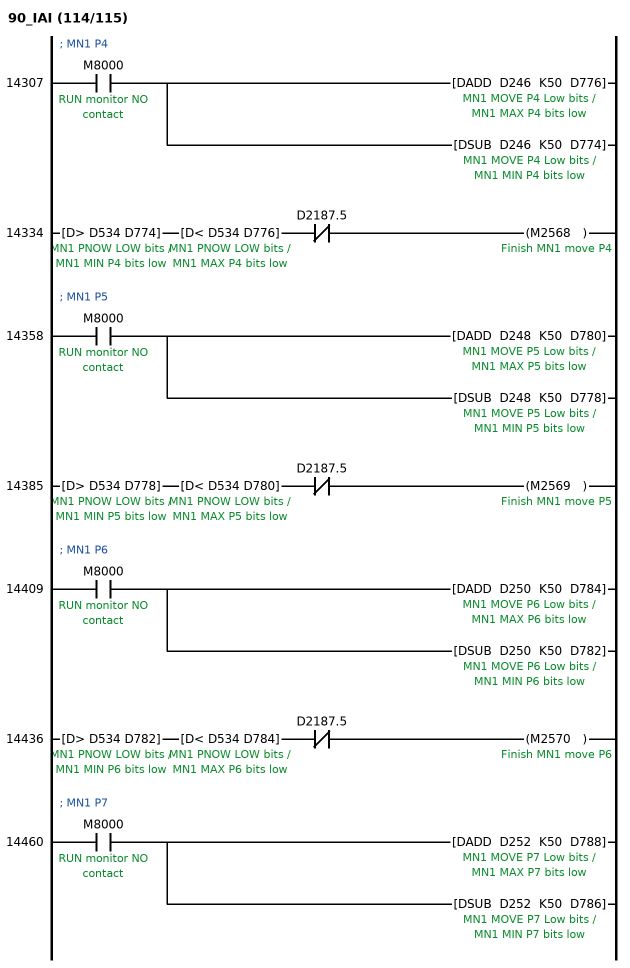
[picture p216: ladder of 90_IAI, rungs at steps 14307 to 14460]
; MN1 P4
14307 LD      M8000  ; RUN monitor NO contact
      DADD    D246 K50 D776  ; MN1 MAX P4 bits low
      DSUB    D246 K50 D774  ; MN1 MIN P4 bits low
14334 LDD>    D534 D774  ; MN1 PNOW LOW bits / MN1 MIN P4 bits low
      ANDD<   D534 D776  ; MN1 PNOW LOW bits / MN1 MAX P4 bits low
      ANI     D2187.5
      OUT     M2568  ; Finish MN1 move P4
; MN1 P5
14358 LD      M8000  ; RUN monitor NO contact
      DADD    D248 K50 D780  ; MN1 MAX P5 bits low
      DSUB    D248 K50 D778  ; MN1 MIN P5 bits low
14385 LDD>    D534 D778  ; MN1 PNOW LOW bits / MN1 MIN P5 bits low
      ANDD<   D534 D780  ; MN1 PNOW LOW bits / MN1 MAX P5 bits low
      ANI     D2187.5
      OUT     M2569  ; Finish MN1 move P5
; MN1 P6
14409 LD      M8000  ; RUN monitor NO contact
      DADD    D250 K50 D784  ; MN1 MAX P6 bits low
      DSUB    D250 K50 D782  ; MN1 MIN P6 bits low
14436 LDD>    D534 D782  ; MN1 PNOW LOW bits / MN1 MIN P6 bits low
      ANDD<   D534 D784  ; MN1 PNOW LOW bits / MN1 MAX P6 bits low
      ANI     D2187.5
      OUT     M2570  ; Finish MN1 move P6
; MN1 P7
14460 LD      M8000  ; RUN monitor NO contact
      DADD    D252 K50 D788  ; MN1 MAX P7 bits low
      DSUB    D252 K50 D786  ; MN1 MIN P7 bits low
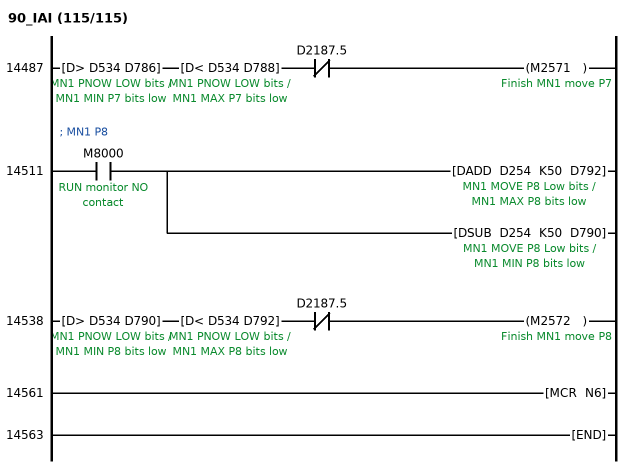
14487 LDD>    D534 D786  ; MN1 PNOW LOW bits / MN1 MIN P7 bits low
      ANDD<   D534 D788  ; MN1 PNOW LOW bits / MN1 MAX P7 bits low
      ANI     D2187.5
      OUT     M2571  ; Finish MN1 move P7
; MN1 P8
14511 LD      M8000  ; RUN monitor NO contact
      DADD    D254 K50 D792  ; MN1 MAX P8 bits low
      DSUB    D254 K50 D790  ; MN1 MIN P8 bits low
14538 LDD>    D534 D790  ; MN1 PNOW LOW bits / MN1 MIN P8 bits low
      ANDD<   D534 D792  ; MN1 PNOW LOW bits / MN1 MAX P8 bits low
      ANI     D2187.5
      OUT     M2572  ; Finish MN1 move P8
14561 MCR     N6
14563 END
END_PROGRAM

PROGRAM 91_Pr_Te
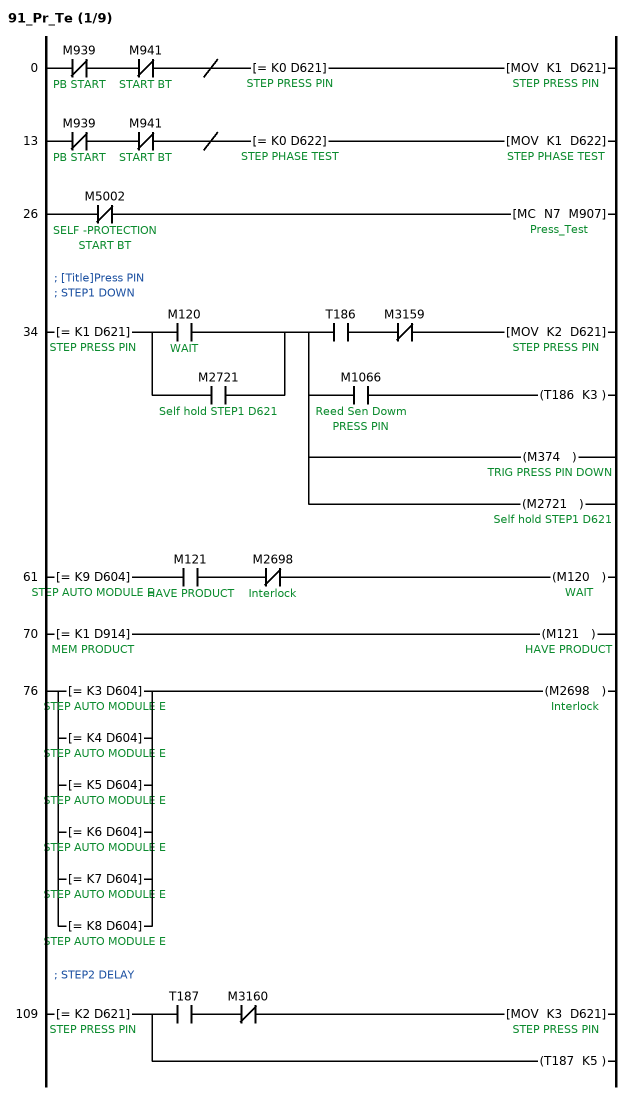
0     LDI     M939  ; PB START
      ANI     M941  ; START BT
      INV
      AND=    K0 D621  ; STEP PRESS PIN
      MOV     K1 D621
13    LDI     M939  ; PB START
      ANI     M941  ; START BT
      INV
      AND=    K0 D622  ; STEP PHASE TEST
      MOV     K1 D622
26    LDI     M5002  ; SELF -PROTECTION START BT
      MC      N7 M907  ; Press_Test
; [Title]Press PIN
; STEP1 DOWN
34    LD=     K1 D621  ; STEP PRESS PIN
      LD      M120  ; WAIT
      OR      M2721  ; Self hold STEP1 D621
      ANB
      MPS
      AND     T186
      ANI     M3159
      MOV     K2 D621
      MRD
      AND     M1066  ; Reed Sen Dowm PRESS PIN
      OUT     T186 K3
      MPP
      OUT     M374  ; TRIG PRESS PIN DOWN
      OUT     M2721  ; Self hold STEP1 D621
61    LD=     K9 D604  ; STEP AUTO MODULE E
      AND     M121  ; HAVE PRODUCT
      ANI     M2698  ; Interlock
      OUT     M120  ; WAIT
70    LD=     K1 D914  ; MEM PRODUCT
      OUT     M121  ; HAVE PRODUCT
76    LD=     K3 D604  ; STEP AUTO MODULE E
      OR=     K4 D604  ; STEP AUTO MODULE E
      OR=     K5 D604  ; STEP AUTO MODULE E
      OR=     K6 D604  ; STEP AUTO MODULE E
      OR=     K7 D604  ; STEP AUTO MODULE E
      OR=     K8 D604  ; STEP AUTO MODULE E
      OUT     M2698  ; Interlock
; STEP2 DELAY
109   LD=     K2 D621  ; STEP PRESS PIN
      MPS
      AND     T187
      ANI     M3160
      MOV     K3 D621
      MPP
      OUT     T187 K5
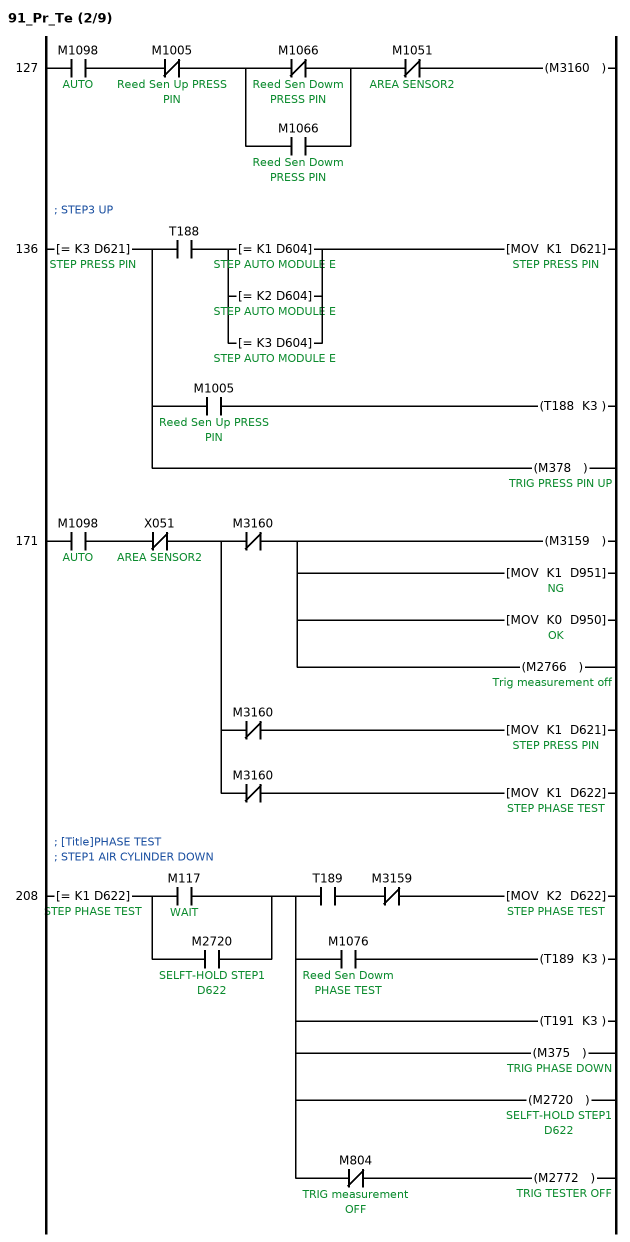
127   LD      M1098  ; AUTO
      ANI     M1005  ; Reed Sen Up PRESS PIN
      LDI     M1066  ; Reed Sen Dowm PRESS PIN
      OR      M1066  ; Reed Sen Dowm PRESS PIN
      ANB
      ANI     M1051  ; AREA SENSOR2
      OUT     M3160
; STEP3 UP
136   LD=     K3 D621  ; STEP PRESS PIN
      MPS
      AND     T188
      LD=     K1 D604  ; STEP AUTO MODULE E
      OR=     K2 D604  ; STEP AUTO MODULE E
      OR=     K3 D604  ; STEP AUTO MODULE E
      ANB
      MOV     K1 D621
      MRD
      AND     M1005  ; Reed Sen Up PRESS PIN
      OUT     T188 K3
      MPP
      OUT     M378  ; TRIG PRESS PIN UP
171   LD      M1098  ; AUTO
      ANI     X051  ; AREA SENSOR2
      MPS
      ANI     M3160
      OUT     M3159
      MOV     K1 D951  ; NG
      MOV     K0 D950  ; OK
      OUT     M2766  ; Trig measurement off
      MRD
      ANI     M3160
      MOV     K1 D621
      MPP
      ANI     M3160
      MOV     K1 D622
; [Title]PHASE TEST
; STEP1 AIR CYLINDER DOWN
208   LD=     K1 D622  ; STEP PHASE TEST
      LD      M117  ; WAIT
      OR      M2720  ; SELFT-HOLD STEP1 D622
      ANB
      MPS
      AND     T189
      ANI     M3159
      MOV     K2 D622
      MRD
      AND     M1076  ; Reed Sen Dowm PHASE TEST
      OUT     T189 K3
      MPP
      OUT     T191 K3
      OUT     M375  ; TRIG PHASE DOWN
      OUT     M2720  ; SELFT-HOLD STEP1 D622
      ANI     M804  ; TRIG measurement OFF
      OUT     M2772  ; TRIG TESTER OFF
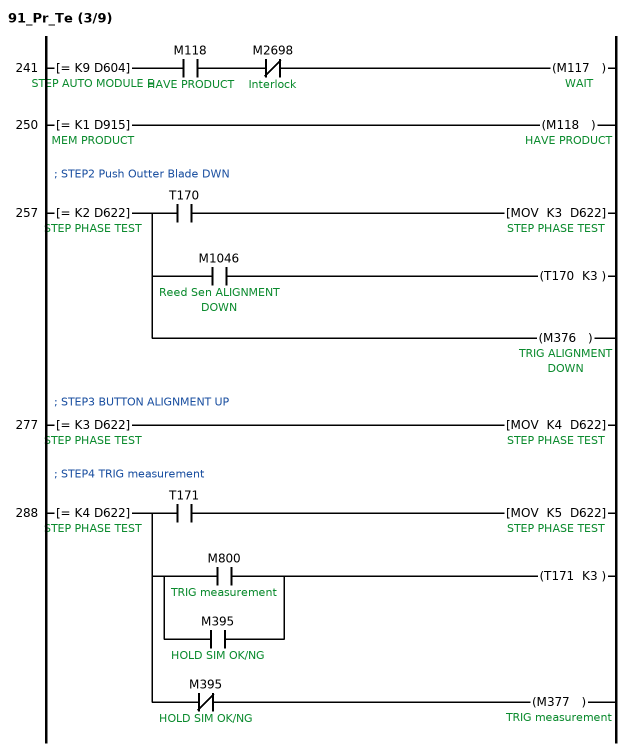
241   LD=     K9 D604  ; STEP AUTO MODULE E
      AND     M118  ; HAVE PRODUCT
      ANI     M2698  ; Interlock
      OUT     M117  ; WAIT
250   LD=     K1 D915  ; MEM PRODUCT
      OUT     M118  ; HAVE PRODUCT
; STEP2 Push Outter Blade DWN
257   LD=     K2 D622  ; STEP PHASE TEST
      MPS
      AND     T170
      MOV     K3 D622
      MRD
      AND     M1046  ; Reed Sen ALIGNMENT DOWN
      OUT     T170 K3
      MPP
      OUT     M376  ; TRIG ALIGNMENT DOWN
; STEP3 BUTTON ALIGNMENT UP
277   LD=     K3 D622  ; STEP PHASE TEST
      MOV     K4 D622
; STEP4 TRIG measurement
288   LD=     K4 D622  ; STEP PHASE TEST
      MPS
      AND     T171
      MOV     K5 D622
      MRD
      LD      M800  ; TRIG measurement
      OR      M395  ; HOLD SIM OK/NG
      ANB
      OUT     T171 K3
      MPP
      ANI     M395  ; HOLD SIM OK/NG
      OUT     M377  ; TRIG measurement
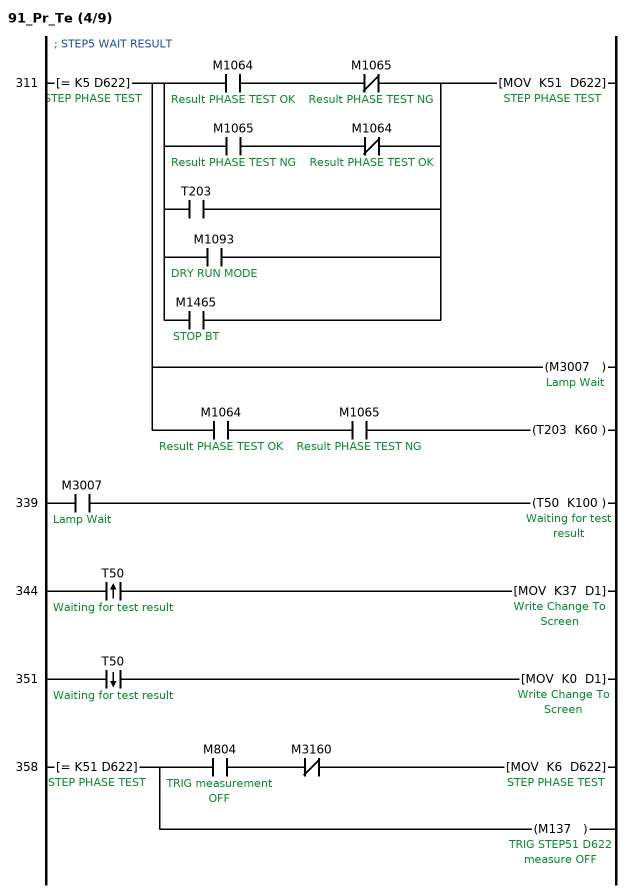
; STEP5 WAIT RESULT
311   LD=     K5 D622  ; STEP PHASE TEST
      MPS
      LD      M1064  ; Result PHASE TEST OK
      ANI     M1065  ; Result PHASE TEST NG
      LD      M1065  ; Result PHASE TEST NG
      ANI     M1064  ; Result PHASE TEST OK
      ORB
      OR      T203
      OR      M1093  ; DRY RUN MODE
      OR      M1465  ; STOP BT
      ANB
      MOV     K51 D622
      MPP
      OUT     M3007  ; Lamp Wait
      AND     M1064  ; Result PHASE TEST OK
      AND     M1065  ; Result PHASE TEST NG
      OUT     T203 K60
339   LD      M3007  ; Lamp Wait
      OUT     T50 K100  ; Waiting for test result
344   LDP     T50  ; Waiting for test result
      MOV     K37 D1  ; Write Change To Screen
351   LDF     T50  ; Waiting for test result
      MOV     K0 D1
358   LD=     K51 D622  ; STEP PHASE TEST
      MPS
      AND     M804  ; TRIG measurement OFF
      ANI     M3160
      MOV     K6 D622
      MPP
      OUT     M137  ; TRIG STEP51 D622 measure OFF
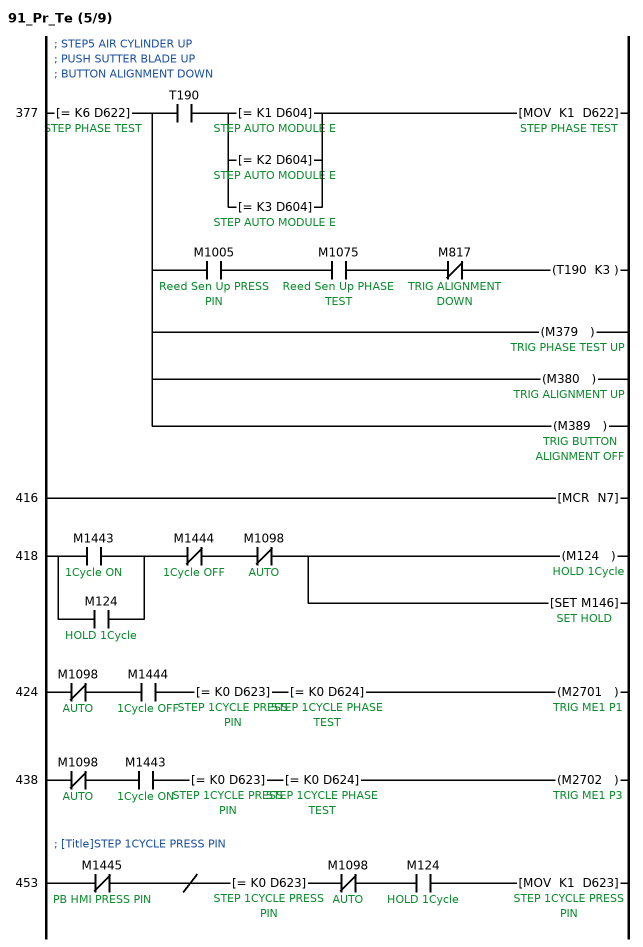
; STEP5 AIR CYLINDER UP
; PUSH SUTTER BLADE UP
; BUTTON ALIGNMENT DOWN
377   LD=     K6 D622  ; STEP PHASE TEST
      MPS
      AND     T190
      LD=     K1 D604  ; STEP AUTO MODULE E
      OR=     K2 D604  ; STEP AUTO MODULE E
      OR=     K3 D604  ; STEP AUTO MODULE E
      ANB
      MOV     K1 D622
      MRD
      AND     M1005  ; Reed Sen Up PRESS PIN
      AND     M1075  ; Reed Sen Up PHASE TEST
      ANI     M817  ; TRIG ALIGNMENT  DOWN
      OUT     T190 K3
      MPP
      OUT     M379  ; TRIG PHASE TEST UP
      OUT     M380  ; TRIG ALIGNMENT UP
      OUT     M389  ; TRIG BUTTON ALIGNMENT OFF
416   MCR     N7
418   LD      M1443  ; 1Cycle ON
      OR      M124  ; HOLD 1Cycle
      ANI     M1444  ; 1Cycle OFF
      ANI     M1098  ; AUTO
      OUT     M124  ; HOLD 1Cycle
      SET     M146  ; SET HOLD
424   LDI     M1098  ; AUTO
      AND     M1444  ; 1Cycle OFF
      AND=    K0 D623  ; STEP 1CYCLE PRESS PIN
      AND=    K0 D624  ; STEP 1CYCLE PHASE TEST
      OUT     M2701  ; TRIG ME1 P1
438   LDI     M1098  ; AUTO
      AND     M1443  ; 1Cycle ON
      AND=    K0 D623  ; STEP 1CYCLE PRESS PIN
      AND=    K0 D624  ; STEP 1CYCLE PHASE TEST
      OUT     M2702  ; TRIG ME1 P3
; [Title]STEP 1CYCLE PRESS PIN
453   LDI     M1445  ; PB HMI PRESS PIN
      INV
      AND=    K0 D623  ; STEP 1CYCLE PRESS PIN
      ANI     M1098  ; AUTO
      AND     M124  ; HOLD 1Cycle
      MOV     K1 D623
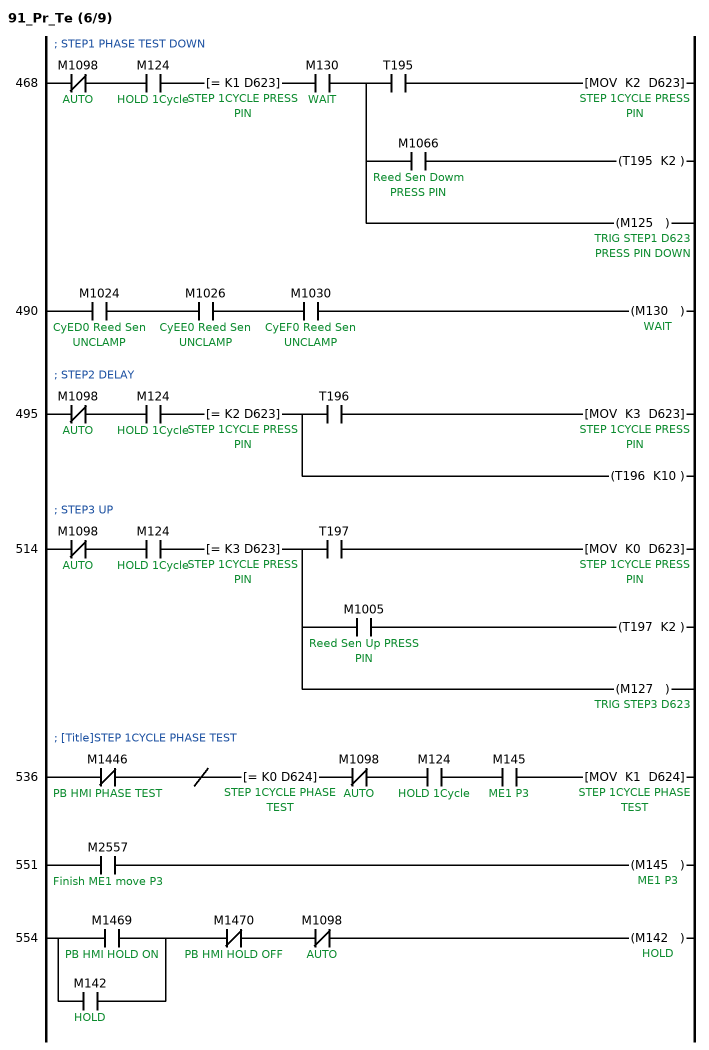
; STEP1 PHASE TEST DOWN
468   LDI     M1098  ; AUTO
      AND     M124  ; HOLD 1Cycle
      AND=    K1 D623  ; STEP 1CYCLE PRESS PIN
      AND     M130  ; WAIT
      MPS
      AND     T195
      MOV     K2 D623
      MRD
      AND     M1066  ; Reed Sen Dowm PRESS PIN
      OUT     T195 K2
      MPP
      OUT     M125  ; TRIG STEP1 D623 PRESS PIN DOWN
490   LD      M1024  ; CyED0 Reed Sen UNCLAMP
      AND     M1026  ; CyEE0 Reed Sen UNCLAMP
      AND     M1030  ; CyEF0 Reed Sen UNCLAMP
      OUT     M130  ; WAIT
; STEP2 DELAY
495   LDI     M1098  ; AUTO
      AND     M124  ; HOLD 1Cycle
      AND=    K2 D623  ; STEP 1CYCLE PRESS PIN
      MPS
      AND     T196
      MOV     K3 D623
      MPP
      OUT     T196 K10
; STEP3 UP
514   LDI     M1098  ; AUTO
      AND     M124  ; HOLD 1Cycle
      AND=    K3 D623  ; STEP 1CYCLE PRESS PIN
      MPS
      AND     T197
      MOV     K0 D623
      MRD
      AND     M1005  ; Reed Sen Up PRESS PIN
      OUT     T197 K2
      MPP
      OUT     M127  ; TRIG STEP3 D623
; [Title]STEP 1CYCLE PHASE TEST
536   LDI     M1446  ; PB HMI PHASE TEST
      INV
      AND=    K0 D624  ; STEP 1CYCLE PHASE TEST
      ANI     M1098  ; AUTO
      AND     M124  ; HOLD 1Cycle
      AND     M145  ; ME1 P3
      MOV     K1 D624
551   LD      M2557  ; Finish ME1 move P3
      OUT     M145  ; ME1 P3
554   LD      M1469  ; PB HMI HOLD ON
      OR      M142  ; HOLD
      ANI     M1470  ; PB HMI HOLD OFF
      ANI     M1098  ; AUTO
      OUT     M142  ; HOLD
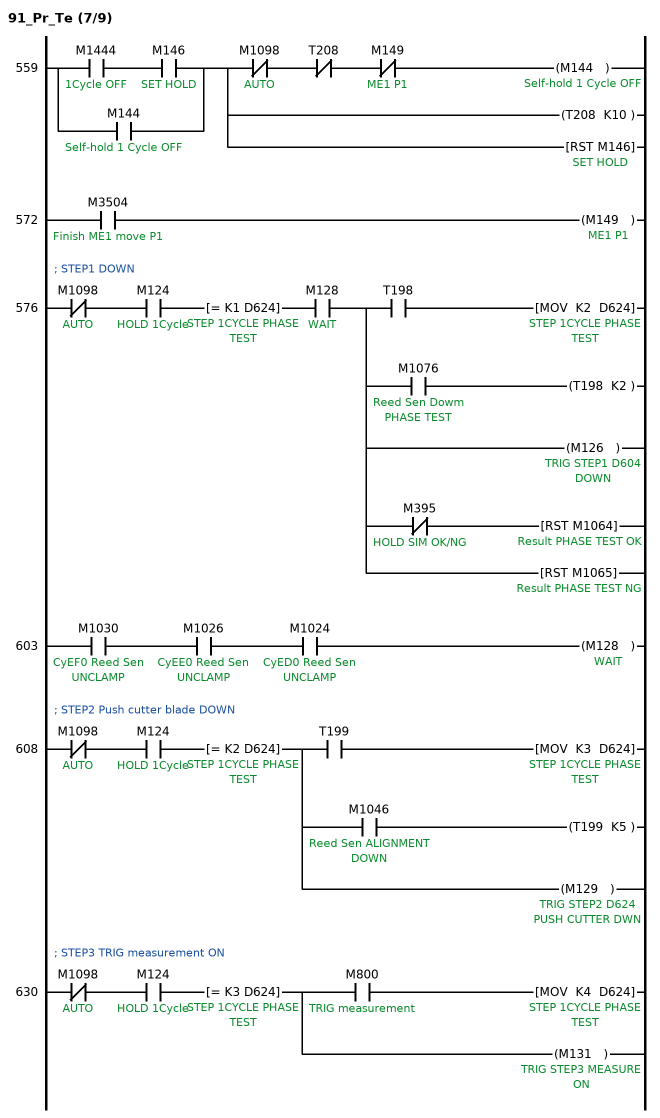
559   LD      M1444  ; 1Cycle OFF
      AND     M146  ; SET HOLD
      OR      M144  ; Self-hold 1 Cycle OFF
      MPS
      ANI     M1098  ; AUTO
      ANI     T208
      ANI     M149  ; ME1 P1
      OUT     M144  ; Self-hold 1 Cycle OFF
      MPP
      OUT     T208 K10
      RST     M146  ; SET HOLD
572   LD      M3504  ; Finish ME1 move P1
      OUT     M149  ; ME1 P1
; STEP1 DOWN
576   LDI     M1098  ; AUTO
      AND     M124  ; HOLD 1Cycle
      AND=    K1 D624  ; STEP 1CYCLE PHASE TEST
      AND     M128  ; WAIT
      MPS
      AND     T198
      MOV     K2 D624
      MRD
      AND     M1076  ; Reed Sen Dowm PHASE TEST
      OUT     T198 K2
      MPP
      OUT     M126  ; TRIG STEP1 D604 DOWN
      MPS
      ANI     M395  ; HOLD SIM OK/NG
      RST     M1064  ; Result PHASE TEST OK
      MPP
      RST     M1065  ; Result PHASE TEST NG
603   LD      M1030  ; CyEF0 Reed Sen UNCLAMP
      AND     M1026  ; CyEE0 Reed Sen UNCLAMP
      AND     M1024  ; CyED0 Reed Sen UNCLAMP
      OUT     M128  ; WAIT
; STEP2 Push cutter blade DOWN
608   LDI     M1098  ; AUTO
      AND     M124  ; HOLD 1Cycle
      AND=    K2 D624  ; STEP 1CYCLE PHASE TEST
      MPS
      AND     T199
      MOV     K3 D624
      MRD
      AND     M1046  ; Reed Sen ALIGNMENT DOWN
      OUT     T199 K5
      MPP
      OUT     M129  ; TRIG STEP2 D624 PUSH CUTTER DWN
; STEP3 TRIG measurement ON
630   LDI     M1098  ; AUTO
      AND     M124  ; HOLD 1Cycle
      AND=    K3 D624  ; STEP 1CYCLE PHASE TEST
      MPS
      AND     M800  ; TRIG measurement
      MOV     K4 D624
      MPP
      OUT     M131  ; TRIG STEP3 MEASURE ON
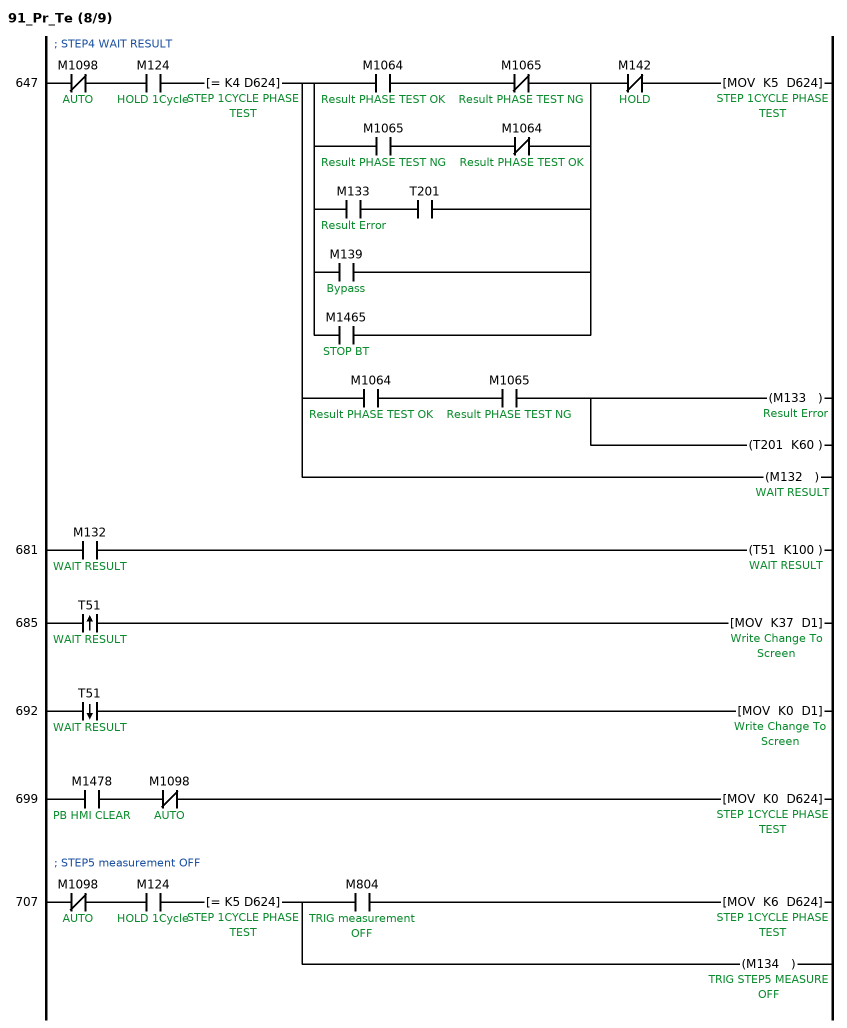
; STEP4 WAIT RESULT
647   LDI     M1098  ; AUTO
      AND     M124  ; HOLD 1Cycle
      AND=    K4 D624  ; STEP 1CYCLE PHASE TEST
      MPS
      LD      M1064  ; Result PHASE TEST OK
      ANI     M1065  ; Result PHASE TEST NG
      LD      M1065  ; Result PHASE TEST NG
      ANI     M1064  ; Result PHASE TEST OK
      ORB
      LD      M133  ; Result Error
      AND     T201
      ORB
      OR      M139  ; Bypass
      OR      M1465  ; STOP BT
      ANB
      ANI     M142  ; HOLD
      MOV     K5 D624
      MRD
      AND     M1064  ; Result PHASE TEST OK
      AND     M1065  ; Result PHASE TEST NG
      OUT     M133  ; Result Error
      OUT     T201 K60
      MPP
      OUT     M132  ; WAIT RESULT
681   LD      M132  ; WAIT RESULT
      OUT     T51 K100  ; WAIT RESULT
685   LDP     T51  ; WAIT RESULT
      MOV     K37 D1
692   LDF     T51  ; WAIT RESULT
      MOV     K0 D1
699   LD      M1478  ; PB HMI CLEAR
      ANI     M1098  ; AUTO
      MOV     K0 D624
; STEP5 measurement OFF
707   LDI     M1098  ; AUTO
      AND     M124  ; HOLD 1Cycle
      AND=    K5 D624  ; STEP 1CYCLE PHASE TEST
      MPS
      AND     M804  ; TRIG measurement OFF
      MOV     K6 D624
      MPP
      OUT     M134  ; TRIG STEP5 MEASURE OFF
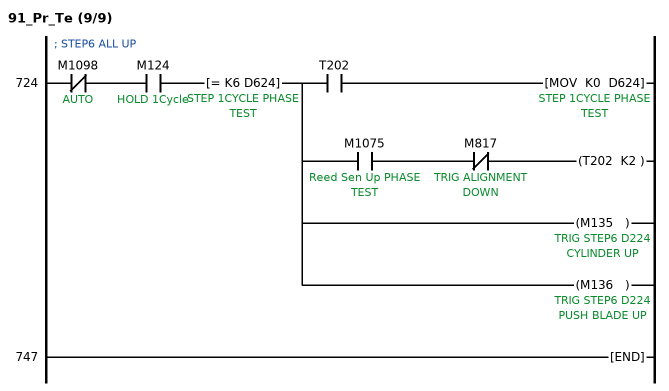
; STEP6 ALL UP
724   LDI     M1098  ; AUTO
      AND     M124  ; HOLD 1Cycle
      AND=    K6 D624  ; STEP 1CYCLE PHASE TEST
      MPS
      AND     T202
      MOV     K0 D624
      MRD
      AND     M1075  ; Reed Sen Up PHASE TEST
      ANI     M817  ; TRIG ALIGNMENT  DOWN
      OUT     T202 K2
      MPP
      OUT     M135  ; TRIG STEP6 D224 CYLINDER UP
      OUT     M136  ; TRIG STEP6 D224 PUSH BLADE UP
747   END
END_PROGRAM

// device comments not shown above
M147  ; ME1 P3
M480  ; 2
M676  ; MUTE LIGHT
M681  ; ALARM RESET
M1018  ; MC2_*ALM
M1048  ; ME1_HOME_OK
M1122  ; REED SW AIR GRIPPER
M1123  ; REED SW AIR GRIPPER
M1128  ; MB3_HOME_OK
M1129  ; MB3_SV
M1138  ; MB3_*ALM
M1148  ; ME1_HOME_OK [CON.2 OUT 14B]
M1149  ; ME1_SV
M1158  ; ME1_*ALM
M1159  ; ME1_HOME_OK SELF-PROTECTION
M1168  ; ALL IAI HOME_OK
M1206  ; TEST
M1217  ; HOME_OK ALL UNCLAMP
M1221  ; XIA = ON
M1222  ; XIB = ON
M1223  ; XIA = ON
M1300  ; HMI PB AIR GRIPPER CLAMP
M1301  ; HMI PB AIR GRIPPER UNCLAMP
M1310  ; PB HMI CyBG Down
M1311  ; PB HMI CyBG UP
M1314  ; PB HMI CyBF Clamp
M1315  ; PB HMI CyBF Unclamp
M1343  ; PB HMI SIDE1 [Y43]
M1406  ; MUTE
M1409  ; PB HMI START FLUX DIP
M1411  ; ALARM RESET
M1413  ; PB HMI RESET STEP HOME
M1418  ; PB HMI Start Flux 1 cycle
M1428  ; PB HMI START NG BLOCK
M1429  ; PB HMI RESTART CON.1
M1460  ; Bypass Result OK/NG ON
M1461  ; Bypass Result OK/NG OFF
M1462  ; HOME BT
M2000  ; PCON 8 AXIS SCAN1
M2001  ; Finsh Mov
M2002  ; Finish MOV
M2150  ; Finish Move
M2216  ; READ SLAVE1 MB1
M2217  ; READ SLAVE2 MB2
M2218  ; READ SLAVE3 MB3
M2219  ; READ SLAVE4 MC1
M2220  ; READ SLAVE5 MC2
M2221  ; READ SLAVE6 MD1
M2222  ; READ SLAVE7 ME1
M2223  ; READ SLAVE8 MN1
M3000  ; PCON 8 AXIS SCAN2
M3562  ; Finish STEP11 D601
M3563  ; Finish STEP12 D601
M4000  ; PCON 8 AXIS SCAN2
M5621  ; ST1 Slave1
M5622  ; ST2 Slave1
M5623  ; ST3 Slave1
M5624  ; ST4 Slave1
M5625  ; ST5 Slave1
M5626  ; ST6 Slave1
M5627  ; ST7 Slave1
M5628  ; JOG- Slave1
M5629  ; JOG+ Slave1
M5634  ; JISL Slave1
M5640  ; DRG1 Slave2
M5661  ; ST1 Slave2
M5662  ; ST2 Slave2
M5663  ; ST3 Slave2
M5664  ; ST4 Slave2
M5665  ; ST5 Slave2
M5666  ; ST6 Slave2
M5667  ; ST7 Slave2
M5668  ; JOG- Slave2
M5669  ; JOG+ Slave2
M5670  ; TEAC Slave2
M5671  ; MOD Slave2
M5674  ; JISL Slave2
M5701  ; ST1 Slave3
M5702  ; ST2 Slave3
M5703  ; ST3 Slave3
M5704  ; ST4 Slave3
M5705  ; ST5 Slave3
M5706  ; ST6 Slave3
M5707  ; ST7 Slave3
M5708  ; JOG- Slave3
M5709  ; JOG+ Slave3
M5714  ; JISL Slave3
M6001  ; Self-hold Bypass Solder Up/Down
D101  ; MB1 MOVE P1 Hight bits
D103  ; MB1 MOVE P2 Hight bits
D105  ; MB1 MOVE P3 Hight bits
D107  ; MB1 MOVE P4 Hight bits
D109  ; MB1 MOVE P5 Hight bits
D111  ; MB1 MOVE P6 Hight bits
D113  ; MB1 MOVE P7 Hight bits
D115  ; MB1 MOVE P8 Hight bits
D117  ; MB1 MOVE P9 Hight bits
D119  ; MB1 MOVE P10 Hight bits
D121  ; MB2 MOVE P1 Hight bits
D123  ; MB2 MOVE P2 Hight bits
D125  ; MB2 MOVE P3 Hight bits
D127  ; MB2 MOVE P4 Hight bits
D129  ; MB2 MOVE P5 Hight bits
D131  ; MB2 MOVE P6 Hight bits
D133  ; MB2 MOVE P7 Hight bits
D135  ; MB2 MOVE P8 Hight bits
D136  ; MB2 MOVE P9 Low bits
D137  ; MB2 MOVE P9 Hight bits
D138  ; MB2 MOVE P10 Low bits
D139  ; MB2 MOVE P10 Hight bits
D141  ; MB3 MOVE P1 Hight bits
D143  ; MB3 MOVE P2 Hight bits
D145  ; MB3 MOVE P3 Hight bits
D147  ; MB3 MOVE P4 Hight bits
D149  ; MB3 MOVE P5 Hight bits
D151  ; MB3 MOVE P6 Hight bits
D153  ; MB3 MOVE P7 Hight bits
D155  ; MB3 MOVE P8 Hight bits
D156  ; MB3 MOVE P9 Low bits
D157  ; MB3 MOVE P9 Hight bits
D158  ; MB3 MOVE P10 Low bits
D159  ; MB3 MOVE P10 Hight bits
D161  ; MC1 MOVE P1 Hight bits
D163  ; MC1 MOVE P2 Hight bits
D165  ; MC1 MOVE P3 Hight bits
D167  ; MC1 MOVE P4 Hight bits
D169  ; MC1 MOVE P5 Hight bits
D171  ; MC1 MOVE P6 Hight bits
D173  ; MC1 MOVE P7 Hight bits
D175  ; MC1 MOVE P8 Hight bits
D176  ; MC1 MOVE P9 Low bits
D177  ; MC1 MOVE P9 Hight bits
D178  ; MC1 MOVE P10 Low bits
D179  ; MC1 MOVE P10 Hight bits
D181  ; MC2 MOVE P1 Hight bits
D183  ; MC2 MOVE P2 Hight bits
D185  ; MC2 MOVE P3 Hight bits
D187  ; MC2 MOVE P4 Hight bits
D189  ; MC2 MOVE P5 Hight bits
D191  ; MC2 MOVE P6 Hight bits
D193  ; MC2 MOVE P7 Hight bits
D195  ; MC2 MOVE P8 Hight bits
D196  ; MC2 MOVE P9 Low bits
D197  ; MC2 MOVE P9 Hight bits
D198  ; MC2 MOVE P10 Low bits
D199  ; MC2 MOVE P10 Hight bits
D201  ; MD1 MOVE P1 Hight bits
D203  ; MD1 MOVE P2 Hight bits
D205  ; MD1 MOVE P3 Hight bits
D207  ; MD1 MOVE P4 Hight bits
D209  ; MD1 MOVE P5 Hight bits
D211  ; MD1 MOVE P6 Hight bits
D213  ; MD1 MOVE P7 Hight bits
D215  ; MD1 MOVE P8 Hight bits
D216  ; MD1 MOVE P9 Low bits
D217  ; MD1 MOVE P9 Hight bits
D218  ; MD1 MOVE P10 Low bits
D219  ; MD1 MOVE P10 Hight bits
D221  ; ME1 MOVE P1 Hight bits
D223  ; ME1 MOVE P2 Hight bits
D225  ; ME1 MOVE P3 Hight bits
D227  ; ME1 MOVE P4 Hight bits
D229  ; ME1 MOVE P5 Hight bits
D231  ; ME1 MOVE P6 Hight bits
D233  ; ME1 MOVE P7 Hight bits
D235  ; ME1 MOVE P8 Hight bits
D236  ; ME1 MOVE P9 Low bits
D237  ; ME1 MOVE P9 Hight bits
D238  ; ME1 MOVE P10 Low bits
D239  ; ME1 MOVE P10 Hight bits
D241  ; MN1 MOVE P1 Hight bits
D243  ; MN1 MOVE P2 Hight bits
D245  ; MN1 MOVE P3 Hight bits
D247  ; MN1 MOVE P4 Hight bits
D249  ; MN1 MOVE P5 Hight bits
D251  ; MN1 MOVE P6 Hight bits
D253  ; MN1 MOVE P7 Hight bits
D255  ; MN1 MOVE P8 Hight bits
D256  ; MN1 MOVE P9 Low bits
D257  ; MN1 MOVE P9 Hight bits
D258  ; MN1 MOVE P10 Low bits
D259  ; MN1 MOVE P10 Hight bits
D260  ; MB1 SPEED P1 Low bits
D261  ; MB1 SPEED P1 Hight bits
D262  ; MB1 SPEED P2 Low bits
D263  ; MB1 SPEED P2 Hight bits
D265  ; MB1 SPEED P3 Hight bits
D266  ; MB1 SPEED P4 Low bits
D267  ; MB1 SPEED P4 Hight bits
D268  ; MB1 SPEED P5 Low bits
D269  ; MB1 SPEED P5 Hight bits
D270  ; MB1 SPEED P6 Low bits
D271  ; MB1 SPEED P6 Hight bits
D272  ; MB1 SPEED P7 Low bits
D273  ; MB1 SPEED P7 Hight bits
D274  ; MB1 SPEED P8 Low bits
D275  ; MB1 SPEED P8 Hight bits
D276  ; MB1 SPEED P9 Low bits
D277  ; MB1 SPEED P9 Hight bits
D279  ; MB1 SPEED P10 Hight bits
D280  ; MB2 SPEED P1 Low bits
D281  ; MB2 SPEED P1 Hight bits
D283  ; MB2 SPEED P2 Hight bits
D285  ; MB2 SPEED P3 Hight bits
D286  ; MB2 SPEED P4 Low bits
D287  ; MB2 SPEED P4 Hight bits
D288  ; MB2 SPEED P5 Low bits
D289  ; MB2 SPEED P5 Hight bits
D291  ; MB2 SPEED P6 Hight bits
D293  ; MB2 SPEED P7 Hight bits
D294  ; MB2 SPEED P8 Low bits
D295  ; MB2 SPEED P8 Hight bits
D296  ; MB2 SPEED P9 Low bits
D297  ; MB2 SPEED P9 Hight bits
D298  ; MB2 SPEED P10 Low bits
D299  ; MB2 SPEED P10 Hight bits
D300  ; MB3 SPEED P1 Low bits
D301  ; MB3 SPEED P1 Hight bits
D302  ; MB3 SPEED P2 Low bits
D303  ; MB3 SPEED P2 Hight bits
D304  ; MB3 SPEED P3 Low bits
D305  ; MB3 SPEED P3 Hight bits
D306  ; MB3 SPEED P4 Low bits
D307  ; MB3 SPEED P4 Hight bits
D308  ; MB3 SPEED P5 Low bits
D309  ; MB3 SPEED P5 Hight bits
D310  ; MB3 SPEED P6 Low bits
D311  ; MB3 SPEED P6 Hight bits
D312  ; MB3 SPEED P7 Low bits
D313  ; MB3 SPEED P7 Hight bits
D314  ; MB3 SPEED P8 Low bits
D315  ; MB3 SPEED P8 Hight bits
D316  ; MB3 SPEED P9 Low bits
D317  ; MB3 SPEED P9 Hight bits
D318  ; MB3 SPEED P10 Low bits
D319  ; MB3 SPEED P10 Hight bits
D320  ; MC1 SPEED P1 Low bits
D321  ; MC1 SPEED P1 Hight bits
D322  ; MC1 SPEED P2 Low bits
D323  ; MC1 SPEED P2 Hight bits
D324  ; MC1 SPEED P3 Low bits
D325  ; MC1 SPEED P3 Hight bits
D326  ; MC1 SPEED P4 Low bits
D327  ; MC1 SPEED P4 Hight bits
D328  ; MC1 SPEED P5 Low bits
D329  ; MC1 SPEED P5 Hight bits
D330  ; MC1 SPEED P6 Low bits
D331  ; MC1 SPEED P6 Hight bits
D332  ; MC1 SPEED P7 Low bits
D333  ; MC1 SPEED P7 Hight bits
D334  ; MC1 SPEED P8 Low bits
D335  ; MC1 SPEED P8 Hight bits
D336  ; MC1 SPEED P9 Low bits
D337  ; MC1 SPEED P9 Hight bits
D338  ; MC1 SPEED P10 Low bits
D339  ; MC1 SPEED P10 Hight bits
D340  ; MC2 SPEED P1 Low bits
D341  ; MC2 SPEED P1 Hight bits
D342  ; MC2 SPEED P2 Low bits
D343  ; MC2 SPEED P2 Hight bits
D344  ; MC2 SPEED P3 Low bits
D345  ; MC2 SPEED P3 Hight bits
D346  ; MC2 SPEED P4 Low bits
D347  ; MC2 SPEED P4 Hight bits
D348  ; MC2 SPEED P5 Low bits
D349  ; MC2 SPEED P5 Hight bits
D350  ; MC2 SPEED P6 Low bits
D351  ; MC2 SPEED P6 Hight bits
D352  ; MC2 SPEED P7 Low bits
D353  ; MC2 SPEED P7 Hight bits
D354  ; MC2 SPEED P8 Low bits
D355  ; MC2 SPEED P8 Hight bits
D356  ; MC2 SPEED P9 Low bits
D357  ; MC2 SPEED P9 Hight bits
D358  ; MC2 SPEED P10 Low bits
D359  ; MC2 SPEED P10 Hight bits
D360  ; MD1 SPEED P1 Low bits
D361  ; MD1 SPEED P1 Hight bits
D362  ; MD1 SPEED P2 Low bits
D363  ; MD1 SPEED P2 Hight bits
D364  ; MD1 SPEED P3 Low bits
D365  ; MD1 SPEED P3 Hight bits
D366  ; MD1 SPEED P4 Low bits
D367  ; MD1 SPEED P4 Hight bits
D368  ; MD1 SPEED P5 Low bits
D369  ; MD1 SPEED P5 Hight bits
D370  ; MD1 SPEED P6 Low bits
D371  ; MD1 SPEED P6 Hight bits
D372  ; MD1 SPEED P7 Low bits
D373  ; MD1 SPEED P7 Hight bits
D374  ; MD1 SPEED P8 Low bits
D375  ; MD1 SPEED P8 Hight bits
D376  ; MD1 SPEED P9 Low bits
D377  ; MD1 SPEED P9 Hight bits
D378  ; MD1 SPEED P10 Low bits
D379  ; MD1 SPEED P10 Hight bits
D380  ; ME1 SPEED P1 Low bits
D381  ; ME1 SPEED P1 Hight bits
D382  ; ME1 SPEED P2 Low bits
D383  ; ME1 SPEED P2 Hight bits
D384  ; ME1 SPEED P3 Low bits
D385  ; ME1 SPEED P3 Hight bits
D386  ; ME1 SPEED P4 Low bits
D387  ; ME1 SPEED P4 Hight bits
D388  ; ME1 SPEED P5 Low bits
D389  ; ME1 SPEED P5 Hight bits
D390  ; ME1 SPEED P6 Low bits
D391  ; ME1 SPEED P6 Hight bits
D392  ; ME1 SPEED P7 Low bits
D393  ; ME1 SPEED P7 Hight bits
D394  ; ME1 SPEED P8 Low bits
D395  ; ME1 SPEED P8 Hight bits
D396  ; ME1 SPEED P9 Low bits
D397  ; ME1 SPEED P9 Hight bits
D398  ; ME1 SPEED P10 Low bits
D399  ; ME1 SPEED P10 Hight bits
D400  ; MN1 SPEED P1 Low bits
D401  ; MN1 SPEED P1 Hight bits
D402  ; MN1 SPEED P2 Low bits
D403  ; MN1 SPEED P2 Hight bits
D404  ; MN1 SPEED P3 Low bits
D405  ; MN1 SPEED P3 Hight bits
D406  ; MN1 SPEED P4 Low bits
D407  ; MN1 SPEED P4 Hight bits
D408  ; MN1 SPEED P5 Low bits
D409  ; MN1 SPEED P5 Hight bits
D410  ; MN1 SPEED P6 Low bits
D411  ; MN1 SPEED P6 Hight bits
D412  ; MN1 SPEED P7 Low bits
D413  ; MN1 SPEED P7 Hight bits
D414  ; MN1 SPEED P8 Low bits
D415  ; MN1 SPEED P8 Hight bits
D416  ; MN1 SPEED P9 Low bits
D417  ; MN1 SPEED P9 Hight bits
D418  ; MN1 SPEED P10 Low bits
D419  ; MN1 SPEED P10 Hight bits
D569  ; MN1 MAX POS hight bit
D571  ; MB1 MIN POS hight bit
D573  ; MB1 MAX POS hight bit
D575  ; MB2 MIN POS hight bit
D577  ; MB2 MAX POS hight bit
D579  ; MB3 MIN POS hight bit
D581  ; MB3 MAX POS hight bit
D583  ; MC1 MIN POS hight bit
D585  ; MC1 MAX POS hight bit
D587  ; MC2 MIN POS hight bit
D589  ; MC2 MAX POS low bit
D591  ; MD1 MIN POS hight bit
D593  ; MD1 MAX POS hight bit
D595  ; ME1 MIN POS hight bit
D597  ; ME1 MAX POS hight bit
D599  ; MN1 MIN POS Hight bit
D711  ; MC2 MIN P1 bits hight
D713  ; MC2 MAX P1 bits hight
D2001  ; LAST SLAVE ID
D2010  ; PNOW[H9000]
D2011  ; PNOW[H9001]
D2013  ; DIPM[H9003]
D2014  ; DOPM[H9004]
D2015  ; DSS1[H9005]
D2016  ; DSS2[H9006]
D2017  ; DSSE[H9007]
D2018  ; STAT1[H9008]
D2019  ; STAT2[H9009]
D3000  ; SLAVE ID SCAN H0D00-H0D01
D3001  ; Last SLAVE ID SCAN H0D00-H0D01
D3010  ; DRG1[H0D00]
D3011  ; DRG2[H0D01]
D4000  ; SLAVE ID SCAN H0D03
D4001  ; LAST SLAVE ID SCAN H0D03
D4010  ; POSR[H0D02]
T112  ; STEP2 D601
